{attribute 'qualified_only'}
VAR_GLOBAL	
	Drive1Settings: ARRAY [0..1] OF XeryonDriveSetting;
	Drive2Settings: ARRAY [0..1] OF XeryonDriveSetting;
	Drive3Settings: ARRAY [0..1] OF XeryonDriveSetting;
	Drive4Settings: ARRAY [0..1] OF XeryonDriveSetting;
END_VAR

(* stored: Version 1.1.0.1, ProductVersion 3.1.4024.11
   GVL GVL: Id {1ca65b75-8ead-4970-ba33-928ed1c6461e} *)
